FUNCTION_BLOCK FB_ItemRegister
VAR_INPUT
	bSignal					: BOOL;
	bReset					: BOOL;
END_VAR
VAR_OUTPUT
	aItemOnTimeRegistry		: ARRAY[0..GVL_Constant.ITEM_ARRAY_SIZE] OF TIME;
	aItemOffTimeRegistry	: ARRAY[0..GVL_Constant.ITEM_ARRAY_SIZE] OF TIME;
	
	nTimeCount				: INT;
END_VAR
VAR
	tTimeOn					: TON;
	tReadTimeOn				: TIME;
	osReadOnTime			: F_TRIG;
	
	tTimeOFF				: TON;
	tReadTimeOff			: TIME;
	osReadOffTime			: R_TRIG;
	
	i						: INT;
END_VAR

IF bSignal THEN
	tTimeOn(IN:=TRUE, PT:=T#5S, ET=>tReadTimeOn);
ELSE
	tTimeOFF(IN:=TRUE, PT:=T#5S, ET=>tReadTimeOff);
END_IF;

//Write on time to array
A_ReadOnTime();

//Write off time to array
A_ReadOffTime();

//Reset array for time registry
A_ResetTimeRegistry();

ACTION A_ReadOffTime:
osReadOffTime(CLK:=bSignal);

IF osReadOffTime.Q THEN
	aItemOffTimeRegistry[nTimeCount] := tReadTimeOff;
	tTimeOff(IN:=FALSE);
END_IF
END_ACTION

ACTION A_ReadOnTime:
osReadOnTime(CLK:=bSignal);

IF osReadOnTime.Q THEN
	aItemOnTimeRegistry[nTimeCount] := tReadTimeOn;
	nTimeCount := nTimeCount +1;
	tTimeOn(IN:=FALSE);
END_IF
END_ACTION

ACTION A_ResetTimeRegistry:
IF bReset THEN
	tTimeOFF(IN:=FALSE);
	tTimeOn(IN:=FALSE);
	
	FOR i := 0 TO nTimeCount DO 
		aItemOffTimeRegistry[i] := T#0S;
		aItemOnTimeRegistry [i] := T#0S;
	END_FOR
	
	nTimeCount := 0;	
	bReset := FALSE;
END_IF
END_ACTION

END_FUNCTION_BLOCK

(* stored: Version 1.1.0.1, ProductVersion 3.1.4024.12
   POU FB_ItemRegister: Id {c0a9bbfd-92cb-44d8-9279-e542f10353df}, SpecialFunc None
   Action A_ReadOffTime: Id {ff391b2f-3597-46da-8b7e-507b7d1c93da}
   Action A_ReadOnTime: Id {eb2f8284-7412-4acb-8aef-a2da25440bbd}
   Action A_ResetTimeRegistry: Id {a95330c9-9324-4e41-9095-d3b44e55e574} *)
